FUNCTION F_EFF_RADIUS : REAL
VAR_INPUT
    RADII : ARRAY[1..10] OF REAL; // Array of Effective Radii
    COUNT : INT;                 //  Number of Lenses
    IF_NONE: REAL;              //  Radius to report if none inserted (-> infinity)
END_VAR
VAR
    INDEX: INT; //Counter for Loop
END_VAR

(*F_EFF_RADIUS

Calculate the effective radius of an array of given lens radii. Non-zero elements
up to the count value are summed in reciprocal space and then inverted to give the
final calculation.
*)

// Initialize
F_EFF_RADIUS := 0.0;

//Sum Reciprocals
WHILE INDEX < COUNT+1 DO
    //Add non-zero element to total
    IF RADII[INDEX] > 0.0 THEN
        F_EFF_RADIUS := F_EFF_RADIUS + 1/RADII[INDEX];
    END_IF
    //Increment
    INDEX := INDEX + 1;
END_WHILE

//Invert if non-zero
/////////////////////
IF F_EFF_RADIUS > 0.0 THEN
    F_EFF_RADIUS := 1/F_EFF_RADIUS;
ELSE
    // B
    F_EFF_RADIUS := IF_NONE;
END_IF

END_FUNCTION

(* stored: Version 1.1.0.1, ProductVersion 3.1.4018.10
   POU F_EFF_RADIUS: Id {f8ea6ca8-8cd4-42de-9ec9-202ffccaf6e8}, SpecialFunc None *)
